FUNCTION_BLOCK FB_setupTrajMoveJ EXTENDS FB_TrajBase
VAR_OUTPUT
END_VAR
VAR
	// move vector in joint space
	m_startPos:Vec5d;
	m_targetPos:Vec5d;
	m_moveDir : Vec5d;
	m_moveDistance :LREAL;
	
	// doubleS planning for move distance
	m_doubleS :FB_BasicDoubleS;
END_VAR

METHOD evaluate : BOOL
VAR_INPUT
	t :LREAL;
END_VAR

VAR_OUTPUT
	jntPos,jntVel, jntAcc :vec5d;
END_VAR
VAR
	q,q_dot,q_ddot :LREAL;
	moveRange :Vec5d;
END_VAR
evaluate:=m_doubleS.evaluate(t,q=>q,q_dot=>q_dot, q_ddot=>q_dot);
IF evaluate =FALSE THEN
	RETURN;
END_IF

vecMultiNum(m_moveDir,q, moveRange);
vecAdd(moveRange, m_startPos,jntPos);
vecMultiNum(m_moveDir,q_dot, jntVel);
vecMultiNum( m_moveDir,q_ddot, jntAcc);
END_METHOD

METHOD init : BOOL
VAR_INPUT
	i_startJntPos :Vec5d;
	i_targetJntPos :Vec5d;
	i_maxJntVel : Vec5d;
	i_maxJntAcc : Vec5d;
	i_maxJntJerk :Vec5d;
END_VAR
VAR 
	i:INT;
	maxV, maxA, maxJ :LREAL;
	q:ARRAY[1..2] OF LREAL;
	v:ARRAY[1..2] OF LREAL;
END_VAR
m_startPos:=i_startJntPos;
m_targetPos:=i_targetJntPos;
vecSub(i_targetJntPos, i_startJntPos, m_moveDir);
m_moveDistance := vecNorm(m_moveDir);

IF(m_moveDistance<g_smallNum) THEN
	vecMultiNum(g_onesVec7d,1/5, m_moveDir);;
ELSE
	vecMultiNum( m_moveDir,1/m_moveDistance, m_moveDir);
END_IF

// determian max vel/acc/jerk
maxV:=g_largeNum;
maxA:=g_largeNum;
maxJ:=g_largeNum;
FOR i :=1 TO 5 DO 
	IF ABS(m_moveDir[i])>g_smallNum THEN
		maxV := MIN (maxV, ABS(i_maxJntVel[i]/m_moveDir[i]));
		maxA := MIN (maxA, ABS(i_maxJntAcc[i]/m_moveDir[i]));
		maxJ := MIN (maxJ, ABS(i_maxJntJerk[i]/m_moveDir[i]));
	END_IF
END_FOR

// planning for moving distance
q[1]:=0;
q[2]:=m_moveDistance;
v[1]:=0;
v[2]:=0;
m_doubleS.init(q,v, maxV, maxA, maxJ);
m_duration:=m_doubleS.duration;
m_isGenerated:=m_doubleS.isGene;
END_METHOD

END_FUNCTION_BLOCK

(* stored: Version 1.1.0.1, ProductVersion 3.1.4024.12
   POU FB_setupTrajMoveJ: Id {cdb6861e-55e5-4dab-9c53-16ea47583316}, SpecialFunc None
   Method evaluate: Id {39c2df8f-cd6f-4472-b175-6ad15a5fa1a1}
   Method init: Id {7907d9c3-586e-4428-a52b-74d1da24d738} *)
